//create working DB
DATA_BLOCK DB2181
STRUCT
START_SEQ:BYTE:=16#1;
END_SEQ:BYTE:=16#2;
SND_COMM_DB:WORD:=16#886;
WRT_COMM_DB:WORD:=16#887;
WRT_COMP_DB:WORD:=16#888;
DAT_RECV_DB:WORD:=16#889;
ACT_1:BOOL:=TRUE;
Mode_1:BOOL:=FALSE;
SND_DB_1:INT:=2182;
SND_ADD_1:INT:=0;
SND_LEN_1:INT:=6;
RCV_DB_1:INT:=2185;
RCV_ADD_1:INT:=0;
RCV_LEN_1:INT:=6;
WD_TIME_1:INT:=3000;
ACT_2:BOOL:=TRUE;
Mode_2:BOOL:=FALSE;
SND_DB_2:INT:=2182;
SND_ADD_2:INT:=8;
SND_LEN_2:INT:=6;
RCV_DB_2:INT:=2185;
RCV_ADD_2:INT:=6;
RCV_LEN_2:INT:=6;
WD_TIME_2:INT:=3000;
VBVer:WORD:=16#2B;   //配置文件版本号
END_STRUCT
BEGIN
END_DATA_BLOCK




//create SND_COMMAND DB
DATA_BLOCK DB2182
STRUCT
SlaveID_1:BYTE:=16#1;
FC_1:BYTE:=16#3;
START_ADD_1:WORD:=16#14;
DATA_NUM_1:WORD:=16#2;
CRC_1:WORD:=16#0;
SlaveID_2:BYTE:=16#2;
FC_2:BYTE:=16#3;
START_ADD_2:WORD:=16#14;
DATA_NUM_2:WORD:=16#2;
CRC_2:WORD:=16#0;
END_STRUCT
BEGIN
END_DATA_BLOCK




//create DAT_COMMAND DB
DATA_BLOCK DB2185
STRUCT
Command_1_STATUS:WORD:=16#0;     //第1条命令的状态，0=正常，1=无响应，2=站号错误，3=命令错误，4=CRC校验错误
Command_1_DATA_1:WORD:=16#0;    //地址40021
Command_1_DATA_2:WORD:=16#0;    //地址40022
Command_2_STATUS:WORD:=16#0;     //第2条命令的状态，0=正常，1=无响应，2=站号错误，3=命令错误，4=CRC校验错误
Command_2_DATA_1:WORD:=16#0;    //地址40021
Command_2_DATA_2:WORD:=16#0;    //地址40022
END_STRUCT
BEGIN
END_DATA_BLOCK
